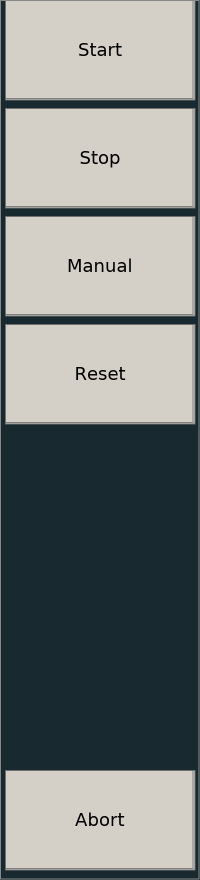
VISUALIZATION NavBarAuto_1  // 200x880
VAR_IN_OUT
	btnStart 		: BOOL;
	btnStop 		: BOOL;
	btnManualMode	: BOOL;
	btnAbort		: BOOL;
	btnReset		: BOOL;
	
	bVisStart 		: BOOL;
	bVisStop		: BOOL;
END_VAR
    Button (5,0 190x100), "Start", input disabled if: bVisStart
        tap btnStart
    Button (5,108 190x100), "Stop", input disabled if: bVisStop
        tap btnStop
    Button (5,770 190x100), "Abort", input disabled if: bVisStart
        tap btnAbort
    Button (5,216 190x100), "Manual", input disabled if: bVisStart
        tap btnManualMode
    Button (5,324 190x100), "Reset", input disabled if: bVisStart
        tap btnReset
END_VISUALIZATION

(* stored: Version 1.1.0.1, ProductVersion 3.1.4024.12
   Visu NavBarAuto_1: Id {57631603-d799-4e0a-9341-85853a61c314} *)
